// TIA Portal V17 export
// export: Created 2025-11-18T11:18:45.8499771Z, ExportSetting WithDefaults, DisplayName Totally Integrated Automation Portal, DisplayVersion V17 Update 8, DisplayName TIA Portal Openness, DisplayVersion V17 Update 8, DisplayName TIA Portal Version Control Interface, DisplayVersion V17, DisplayName STEP 7 Professional, DisplayVersion V17 Update 8, DisplayName STEP 7 Safety, DisplayVersion V17 Update 6, DisplayName WinCC Advanced, DisplayVersion V17 Update 8
DATA_BLOCK "PLC_PLC_Connection_DB"   // DB9
VERSION : 0.1
// stored: AutoNumber true, DBAccessibleFromOPCUA true, InstanceOfName PLC_VLC_Connection_TCP-IP, InstanceOfType FB
"PLC_VLC_Connection_TCP-IP"
   // VAR_INPUT
   //    xFirstScan : Bool;
   //    xAlwaysTRUE : Bool;
   //    xDataReceiveOn : Bool;
   // END_VAR
   // VAR_OUTPUT
   //    Connection_OK : Bool;
   //    Connected : Bool;
   //    Started : Bool;
   //    Paused : Bool;
   //    EndOfFile : Bool;
   // END_VAR
   // VAR_IN_OUT
   //    xSendRequest : Bool;
   //    xCommandStart : Bool;
   //    xCommandStop : Bool;
   //    xCommandReset : Bool;
   //    xCommandPause : Bool;
   //    xCommandResume : Bool;
   //    xCommandRewind0 : Bool;
   //    xCommandRewindX : Bool;
   //    xReconnect : Bool;
   // END_VAR
   // VAR
   //    TCON_Instance { S7_SetPoint := 'True'} : TCON;
   //    TCON : Struct
   //       REC : Bool;
   //       DONE : Bool;
   //       BUSY : Bool;
   //       ERROR : Bool;
   //       DONE_Memo : Bool;
   //       STATUS : Word;
   //    END_STRUCT;
   //    TDISCON : Struct
   //       REQ : Bool;
   //       DONE : Bool;
   //       BUSY : Bool;
   //       ERROR : Bool;
   //       STATUS : Word;
   //    END_STRUCT;
   //    TSEND : Struct
   //       REQ : Bool;
   //       DONE : Bool;
   //       BUSY : Bool;
   //       ERROR : Bool;
   //       DONE_Memo : Bool;
   //       STATUS : Word;
   //    END_STRUCT;
   //    TRCV : Struct
   //       EN_R : Bool;
   //       NDR : Bool;
   //       BUSY : Bool;
   //       ERROR : Bool;
   //       STATUS : Word;
   //       RCVD_LENGTH : UDInt;
   //    END_STRUCT;
   //    TDISCON_DB { S7_SetPoint := 'True'} : TDISCON;
   //    TSEND_Instance { S7_SetPoint := 'True'} : TSEND;
   //    TRCV_Instance { S7_SetPoint := 'True'} : TRCV;
   //    Variables : Struct
   //       ConnectRequest : Bool;
   //       DisconnectRequest : Bool;
   //       Reconect : Bool;
   //       SendString : String;
   //       DataToSend : String;
   //       Heartbeat0 : Bool;
   //       Heartbeat1 : Bool;
   //       Heartbeat_ConnectionOK : Bool;
   //       Receive : Array[0..20] of Char;
   //       ReceivedString : String;
   //    END_STRUCT;
   //    Pulses { S7_SetPoint := 'True'} : Array[0..10] of Bool;
   //    IEC_Timer_SendData { S7_SetPoint := 'True'} : TP_TIME;
   //    IEC_Timer_SendRequestToLong { S7_SetPoint := 'True'} : TON_TIME;
   //    IEC_TimerReconnect { S7_SetPoint := 'True'} : TON_TIME;
   //    IEC_Timer_ReadDelayAfterConnect { S7_SetPoint := 'True'} : TON_TIME;
   //    TON_HB_1 { S7_SetPoint := 'True'} : TON_TIME;
   //    TON_HB_2 { S7_SetPoint := 'True'} : TON_TIME;
   //    TON_HB_3 { S7_SetPoint := 'True'} : TON_TIME;
   //    ReconnectTimer { S7_SetPoint := 'True'} : TON_TIME;
   //    RecoonectTimer2 { S7_SetPoint := 'True'} : TON_TIME;
   //    pulse : Bool;
   //    pulse2 : Bool;
   //    resetTimera : Bool;
   //    pulse3 : Bool;
   // END_VAR
BEGIN
END_DATA_BLOCK
